TYPE DigitalInput :
STRUCT
	in AT %I*	:	BIT;
END_STRUCT
END_TYPE

(* stored: Version 1.1.0.1, ProductVersion 3.1.4020.12
   DUT DigitalInput: Id {bdb41fff-0c80-427a-8ccd-51cd938fd963} *)
